FUNCTION FC_InitializeNameAsNeeded	// Can be used to initialize the given name of a component
VAR_INPUT
	iInit:	T_SHORT_STR;		// Initial value
END_VAR
VAR_IN_OUT
	ioMonitor:	T_SHORT_STR;	// String to be monitored
END_VAR

IF (NOT FC_IsBaseNameDefined(ioMonitor)) THEN
	ioMonitor := iInit;
END_IF

END_FUNCTION

(* stored: Version 1.1.0.1, ProductVersion 3.1.4026.18
   POU FC_InitializeNameAsNeeded: Id {a8071e54-1644-4f0f-99f9-dc4e1f04b3b7}, SpecialFunc None *)
